Staubli VAL3: create.pgx

public program create(num x_nEncNum, string x_sTask)
begin
  call init(x_nEncNum,x_sTask)
  taskCreate sTASK,100,encoder()
end
